FUNCTION_BLOCK PneumaticInsertionEIP
VAR_INPUT
	enable : BOOL;
END_VAR
VAR_OUTPUT
	slider : ClearLinkMC;
	screw : AirPiston;
	
	contact : BOOL;
	
	home : BOOL;
	ready : BOOL;
	busy : BOOL;
	error : BOOL;
	
	sliderPos : LREAL;
END_VAR

slider(
	bEnable:= enable, 
	pulse=> , 
	outputRegister=> , 
	brakeRelease=> , 
	A=> , 
	B=> , 
	clear=> , 
	contactSensor=> , 
	home=> , 
	outerLimit=> , 
	innerLimit=> , 
	hlfb=> , 
	homingComplete=> , 
	Busy=> , 
	Error=> , 
	targetPos=> );

sliderPos := slider.CurrentPosition;	
	
screw(
	bEnable:= enable,
	valveExtend=> , 
	valveRetract=> , 
	contactSensor=> , 
	home=> , 
	innerLimit=> , 
	Busy=> , 
	Error=> , 
	homingComplete=> );
	
home := screw.AtHome AND slider.AtHome;
busy := slider.Busy OR screw.Busy;
error := slider.Error OR screw.Error;

METHOD homingSequence : BOOL
(*
IF NOT slider.homeSet THEN
	slider.homingSequence();
END_IF
*)
IF NOT screw.homingComplete THEN
	screw.homingSequence();
END_IF

homingSequence := (*slider.homeSet AND*) screw.homingComplete;
END_METHOD

METHOD press : BOOL
VAR_INPUT
	//direction : BOOL; //direction (F = inwards, T = outwards)
	//distance : DINT;
END_VAR
press := screw.extend();
END_METHOD

METHOD release : BOOL
VAR_INPUT
END_VAR
release := screw.retract();
END_METHOD

METHOD slideAbsolute : BOOL
VAR_INPUT
	targetPos : REAL;
END_VAR
slideAbsolute := slider.moveAbsolute(newTarget:= targetPos);
END_METHOD

METHOD slideContinuous : BOOL
VAR_INPUT
	direction : MC_Direction;
END_VAR
slideContinuous := slider.moveContinuous(direction := direction);
END_METHOD

END_FUNCTION_BLOCK

(* stored: Version 1.1.0.1, ProductVersion 3.1.4024.11
   POU PneumaticInsertionEIP: Id {60eb499d-0a9f-498e-8b27-5c86a4039353}, SpecialFunc None
   Method homingSequence: Id {74aa10a4-d54f-4feb-b7ba-b023029d51d3}
   Method press: Id {6d696dd3-7676-4d35-8862-76ab2dec8fa9}
   Method release: Id {df15fb9e-4c1d-4296-8fe1-9b7e99ff36b4}
   Method slideAbsolute: Id {7157da18-36ff-410d-8d76-ea3b77265589}
   Method slideContinuous: Id {1746ade4-dd8f-4b66-9808-8ec1918d6c35} *)
